FUNCTION_BLOCK FB_BoolTrigger EXTENDS FB_Base		// Detects rising and falling edges on the input
VAR_INPUT
	iIn:			BOOL;
END_VAR
VAR_OUTPUT
	oRtrig:			BOOL;
	oFtrig:			BOOL;
	oChanged:		BOOL;
END_VAR
VAR
	rTrig:			R_TRIG;
	fTrig:			F_TRIG;
END_VAR

rTrig(CLK := iIn, Q => oRtrig);
fTrig(CLK := iIn, Q => oFtrig);

oChanged := oRtrig OR oFtrig;

END_FUNCTION_BLOCK

(* stored: Version 1.1.0.1, ProductVersion 3.1.4026.18
   POU FB_BoolTrigger: Id {b74a10c5-4bda-4e78-bcf7-dc9161fe573f}, SpecialFunc None *)
